// TIA Portal V16 export
// export: Created 2024-12-03T15:41:42.2460899Z, ExportSetting WithDefaults, DisplayName Totally Integrated Automation Portal, DisplayVersion V16 Update 6, DisplayName TIA Portal Version Control Interface, DisplayVersion V16 Update 2, DisplayName TIA Portal Openness, DisplayVersion V16 Update 6, DisplayName TIA Portal Teamcenter Gateway, DisplayVersion V16, DisplayName SINAMICS Startdrive Advanced, DisplayVersion V16 Update 5, DisplayName SINAMICS Startdrive G130, G150, S120, S150, SINAMICS MV, S210, DisplayVersion V16 Update 5, DisplayName SINAMICS Startdrive G110M, G120, G120C, G120D, G120P, G115D, DisplayVersion V16 Update 5, DisplayName STEP 7 Professional, DisplayVersion V16 Update 6, DisplayName STEP 7 Safety, DisplayVersion V16, DisplayName WinCC Advanced / Unified PC, DisplayVersion V16 Update 6
FUNCTION_BLOCK "CylinderController"   // FB5, SCL
{ S7_Optimized_Access := 'FALSE' }
VERSION : 0.1
// stored: AutoNumber true, IsIECCheckEnabled false, SetENOAutomatically false, UDAEnableTagReadback false
   VAR_INPUT
      I_AlwaysAuto : Bool;
      I_DbName : String := '"Cylinders_DB".';
      I_Interlock : Bool;
      I_CylinderInFeedBack : Bool;   // Cylinder is in feedback
      I_CylinderOutFeedBack : Bool;   // Cylinder is out feedback
   END_VAR
   VAR_OUTPUT
      O_CmdIn : Bool;
      O_CmdOut : Bool;
   END_VAR
   VAR_IN_OUT
      IO_Cyl : "Cylinder_UDT";
   END_VAR
   VAR DB_SPECIFIC
      feedBackTimeIn : TON_TIME;
      feedBackTimeOut : TON_TIME;
      TimeIn { S7_SetPoint := 'True'} : TON_TIME;
      TimeOut { S7_SetPoint := 'True'} : TON_TIME;
      Info { S7_SetPoint := 'True'} : "AlarmInfo_UDT";
   END_VAR
   VAR
      alarmNotIn { S7_SetPoint := 'True'} : Program_Alarm;
   END_VAR
   VAR DB_SPECIFIC
      ZoneInfo { ExternalAccessible := 'False'; ExternalVisible := 'False'; ExternalWritable := 'False'} : "ZoneInfo";
   END_VAR
   VAR
      alarmNotOut { S7_SetPoint := 'True'} : Program_Alarm;
   END_VAR
   VAR_TEMP
      T_AppState : "ApplicationState_UDT";
   END_VAR
BEGIN
   #ZoneInfo := "ApplicationState_DB".ZoneNames[#IO_Cyl.Zone];
   #T_AppState := "ApplicationState_DB".Appstate[#ZoneInfo.AppStateIndex];
   REGION Detect position

       #feedBackTimeIn(IN:=#I_CylinderInFeedBack,
                       PT:=#IO_Cyl.Settings.feedBackInDelay);

       #feedBackTimeOut(IN:=#I_CylinderOutFeedBack,
                        PT:=#IO_Cyl.Settings.feedBackOutDelay);

       //Cylinder out
       IF NOT #feedBackTimeIn.Q AND #feedBackTimeOut.Q THEN
           #IO_Cyl.Status.Position := 1;
       END_IF;

       //Cylinder in
       IF #feedBackTimeIn.Q AND NOT #feedBackTimeOut.Q THEN
           #IO_Cyl.Status.Position := -1;
       END_IF;

       //Cylinder traveling
       IF NOT #feedBackTimeIn.Q AND NOT #feedBackTimeOut.Q THEN
           #IO_Cyl.Status.Position := 0;
       END_IF;

   END_REGION

   REGION Interlock

       #IO_Cyl.Status.Interlocked := #I_Interlock OR #IO_Cyl.Cmd.Interlock;
       #IO_Cyl.Status.status.%X0 := #IO_Cyl.Status.Interlocked;

   END_REGION

   REGION Manual MODe active

       #IO_Cyl.Status.ManualModeActive := #T_AppState.States.ManualModeActivated.State AND NOT #I_AlwaysAuto;
       #IO_Cyl.Status.status.%X1 := #IO_Cyl.Status.ManualModeActive;

   END_REGION

   REGION Copy commands

       #IO_Cyl.Status.ManualCommandsDisabled := 0;

       //Clear commands
       IF NOT #IO_Cyl.Settings.CopyCommands THEN
           #O_CmdOut := 0;
           #O_CmdIn := 0;
       END_IF;

       REGION AUTO MODE

           IF #T_AppState.States.AutoModeActivated.State OR #I_AlwaysAuto THEN
               IF NOT #IO_Cyl.Cmd.Interlock THEN
                   IF #IO_Cyl.Settings.CylinderType = 1 OR #IO_Cyl.Settings.CylinderType = 2 THEN
                       #O_CmdOut := 0;
                       #O_CmdIn := 0;
                       IF #IO_Cyl.Cmd.OutAuto THEN
                           #IO_Cyl.Cmd.InAuto := FALSE;
                           #O_CmdOut := #IO_Cyl.Cmd.OutAuto;
                           #O_CmdIn := NOT #O_CmdOut;
                       END_IF;
                       IF #IO_Cyl.Cmd.InAuto THEN
                           #IO_Cyl.Cmd.OutAuto := FALSE;
                           #O_CmdIn := #IO_Cyl.Cmd.InAuto;
                           #O_CmdOut := NOT #O_CmdIn;
                       END_IF;
                   ELSE
                       #O_CmdOut := #IO_Cyl.Cmd.OutAuto;
                       #O_CmdIn := #IO_Cyl.Cmd.InAuto;
                   END_IF;
               END_IF;

           END_IF;

       END_REGION

       REGION MANUAL MODE

           IF NOT #T_AppState.States.ManualModeActivated.State AND NOT #I_AlwaysAuto THEN
               IF NOT #IO_Cyl.Settings.CopyCommands THEN
                   #IO_Cyl.Cmd.OutManual := 0;
                   #IO_Cyl.Cmd.InManual := 0;
               END_IF;
               #IO_Cyl.Status.ManualCommandsDisabled := 1;
           END_IF;

           IF #T_AppState.States.ManualModeActivated.State THEN
               IF NOT #IO_Cyl.Cmd.Interlock THEN
                   IF #IO_Cyl.Cmd.OutManualHMI AND #IO_Cyl.Settings.EnableManualOut THEN
                       #IO_Cyl.Cmd.OutManual := 1;
                       #IO_Cyl.Cmd.InManual := 0;
                   END_IF;

                   IF #IO_Cyl.Cmd.InManualHMI AND #IO_Cyl.Settings.EnableManualIn THEN
                       #IO_Cyl.Cmd.InManual := 1;
                       #IO_Cyl.Cmd.OutManual := 0;
                   END_IF;
               ELSE
                   #IO_Cyl.Cmd.InManual := #O_CmdIn;
                   #IO_Cyl.Cmd.OutManual := #O_CmdOut;
               END_IF;

               IF #IO_Cyl.Cmd.InManualHMI OR #IO_Cyl.Cmd.OutManualHMI THEN
                   #IO_Cyl.Cmd.InManualHMI := 0;
                   #IO_Cyl.Cmd.OutManualHMI := 0;
               END_IF;

               #O_CmdOut := #IO_Cyl.Cmd.OutManual;
               #O_CmdIn := #IO_Cyl.Cmd.InManual;
           END_IF;

       END_REGION

       REGION copy commands
           IF #IO_Cyl.Settings.CopyCommands THEN

               IF #T_AppState.States.ManualModeActivated.State THEN
                   #IO_Cyl.Cmd.InAuto := #IO_Cyl.Cmd.InManual;
                   #IO_Cyl.Cmd.OutAuto := #IO_Cyl.Cmd.OutManual;
               END_IF;

               IF #T_AppState.States.AutoModeActivated.State THEN
                   #IO_Cyl.Cmd.InManual := #IO_Cyl.Cmd.InAuto;
                   #IO_Cyl.Cmd.OutManual := #IO_Cyl.Cmd.OutAuto;
               END_IF;

               END_IF;

       END_REGION

       REGION DISABLE COMMANDS ON ERROR
           IF NOT #T_AppState.States.EmergencyOk.State OR
               (#IO_Cyl.Alarms.Status > 0 AND NOT #IO_Cyl.Settings.CmdOnError)
               OR #IO_Cyl.Status.Interlocked THEN

               #IO_Cyl.Cmd.OutManualHMI := 0;
               #IO_Cyl.Cmd.InManualHMI := 0;
               #O_CmdOut := 0;
               #O_CmdIn := 0;
               #IO_Cyl.Status.ManualCommandsDisabled := 1;

           END_IF;
       END_REGION

   END_REGION

   REGION OBJECT NAME

       IF NOT #Info.init OR #Info.info = '' OR #IO_Cyl.Name = '' OR "HMI_DB".ReloadSettings.signal THEN
           #IO_Cyl.Name := "buildObjectName"(I_Symbolname := GetSymbolName(variable := #IO_Cyl, size := 100));
           #Info.info := "buildAlarmInfo"(I_ObjectName := #IO_Cyl.Name, I_ZoneIndex := #ZoneInfo.AppStateIndex, I_ZoneName := #ZoneInfo.ZoneName);
           #Info.init := true;
       END_IF;

   END_REGION

   REGION Alarms

       REGION Alarms bistabiel

           IF #IO_Cyl.Settings.CylinderType = 0 THEN

               #TimeIn(IN := #O_CmdIn AND NOT #I_CylinderInFeedBack,
                         PT := #IO_Cyl.Settings.CylinderInTime);

               IF #TimeIn.Q THEN
                   #IO_Cyl.Alarms.NotIn.Active := true;
               END_IF;

               #TimeOut(IN := #O_CmdOut AND NOT #I_CylinderOutFeedBack,
                          PT := #IO_Cyl.Settings.CylinderOutTime);

               IF #TimeOut.Q THEN
                   #IO_Cyl.Alarms.NotOut.Active := true;
               END_IF;

           END_IF;


       END_REGION

       REGION Alarms mono in

           IF #IO_Cyl.Settings.CylinderType = 1 THEN

               #TimeIn(IN := NOT #O_CmdOut AND NOT #I_CylinderInFeedBack,
                         PT := #IO_Cyl.Settings.CylinderInTime);

               IF #TimeIn.Q THEN
                   #IO_Cyl.Alarms.NotIn.Active := true;
               END_IF;

               #TimeOut(IN := #O_CmdOut AND NOT #I_CylinderOutFeedBack,
                          PT := #IO_Cyl.Settings.CylinderOutTime);

               IF #TimeOut.Q THEN
                   #IO_Cyl.Alarms.NotOut.Active := true;
               END_IF;

           END_IF;


       END_REGION

       REGION Alarms mono out

           IF #IO_Cyl.Settings.CylinderType = 2 THEN

               #TimeIn(IN := #O_CmdIn AND NOT #I_CylinderInFeedBack,
                         PT := #IO_Cyl.Settings.CylinderInTime);

               IF #TimeIn.Q THEN
                   #IO_Cyl.Alarms.NotIn.Active := true;
               END_IF;

               #TimeOut(IN := NOT #O_CmdIn AND NOT #I_CylinderOutFeedBack,
                          PT := #IO_Cyl.Settings.CylinderOutTime);

               IF #TimeOut.Q THEN
                   #IO_Cyl.Alarms.NotOut.Active := true;
               END_IF;

           END_IF;

       END_REGION

       REGION PROGRAM ALARM

           #alarmNotIn(SIG := #IO_Cyl.Alarms.NotIn.Active, SD_1 := #ZoneInfo.ZoneName, SD_2 := #IO_Cyl.Name, SD_3 := #Info.info);
           #alarmNotOut(SIG := #IO_Cyl.Alarms.NotOut.Active, SD_1 := #ZoneInfo.ZoneName, SD_2 := #IO_Cyl.Name, SD_3 := #Info.info);

       END_REGION

       REGION Create alarm status

           #IO_Cyl.Alarms.Status.%X0 := #IO_Cyl.Alarms.NotIn.Active;
           #IO_Cyl.Alarms.Status.%X1 := #IO_Cyl.Alarms.NotOut.Active;

       END_REGION

       IF #IO_Cyl.Alarms.Status > 0 THEN
           "ApplicationState_DB".Appstate[#ZoneInfo.AppStateIndex].Alarms.AlarmActiveInternalPLC := TRUE;
       END_IF;

   END_REGION

   REGION Reset 

       IF "Inputs_DB".Reset_System.State THEN
           RESET_TIMER(#TimeIn);
           RESET_TIMER(#TimeOut);
           #IO_Cyl.Alarms.NotIn.Active := 0;
           #IO_Cyl.Alarms.NotOut.Active := 0;
       END_IF;

   END_REGION
END_FUNCTION_BLOCK
